// TIA Portal project "Lab1" (V15)

(* hardware
DEVICE "S7-1200 station_1"  S7-1200 Station
   slot 0: "Rack_0"  S7-1200 Rack  Rack  V1.0
   slot 1: "PLC_1"  CPU 1214C AC/DC/Rly  6ES7 214-1BG40-0XB0  V4.2
*)

// ===== PLC "PLC_1"  CPU 1214C AC/DC/Rly =====

VAR_GLOBAL   // PLC tag table "Default tag table"
   "Start_NC" AT %I0.0 : Bool;
   "Manual_NO" AT %I0.2 : Bool;
   "Auto_NO" AT %I0.3 : Bool;
   "Stop_NC" AT %I0.4 : Bool;
   "SigSklop_NC" AT %I0.6 : Bool;
   "Bimetal_NC" AT %I0.7 : Bool;
   "Prekostruj_NO" AT %I1.0 : Bool;
   "Kontaktor_NO" AT %I1.1 : Bool;
   "Zelena" AT %Q0.0 : Bool;
   "Crvena" AT %Q0.1 : Bool;
   "Kontaktor" AT %Q0.2 : Bool;
   "Clock_Byte" AT %MB53 : Byte;
   "Clock_10Hz" AT %M53.0 : Bool;
   "Clock_5Hz" AT %M53.1 : Bool;
   "Clock_2.5Hz" AT %M53.2 : Bool;
   "Clock_2Hz" AT %M53.3 : Bool;
   "Clock_1.25Hz" AT %M53.4 : Bool;
   "Clock_1Hz" AT %M53.5 : Bool;
   "Clock_0.625Hz" AT %M53.6 : Bool;
   "Clock_0.5Hz" AT %M53.7 : Bool;
   "Blink" AT %M3.2 : Bool;
   "Blink_FF" AT %M3.1 : Bool;
   "Blink_Pulse" AT %M3.0 : Bool;
   "Auto_Stanje_FF" AT %M2.0 : Bool;
   "Greska" AT %M0.4 : Bool;
   "Greska_Bimetal" AT %M0.0 : Bool;
   "Greska_Prekostruj" AT %M0.1 : Bool;
   "Greska_Kontaktor" AT %M0.2 : Bool;
   "Greska_Svestop" AT %M0.3 : Bool;
   "Cekamo" AT %M2.2 : Bool;
   "Blink_Cnt_Greska_Pos" AT %M3.3 : Bool;
   "Blink_FF_Greska_Pos" AT %M3.4 : Bool;
   "OFF_NO" AT %M2.1 : Bool;
   "Bimetal_FF" AT %M1.0 : Bool;
   "Prekostruj_FF" AT %M1.1 : Bool;
   "Svestop_FF" AT %M1.3 : Bool;
   "GKontaktor_FF" AT %M1.2 : Bool;
   "Cekamo_Trig_P" AT %M2.3 : Bool;
   "Cekamo_Trig_N" AT %M2.4 : Bool;
   "Ocekivani_Kontaktor" AT %M2.5 : Bool;
END_VAR

// folder: System blocks/Program resources

DATA_BLOCK "Counter_Blink"   // DB1
{ S7_Optimized_Access := 'TRUE' }
AUTHOR : Simatic
FAMILY : IEC
NAME : CNTR
VERSION : 1.0
// stored: InstanceOfName IEC_COUNTER
"IEC_COUNTER"
BEGIN
END_DATA_BLOCK

DATA_BLOCK "Timer_Start"   // DB2
{ S7_Optimized_Access := 'TRUE' }
AUTHOR : Simatic
FAMILY : IEC
NAME : IEC_TMR
VERSION : 1.0
// stored: InstanceOfName IEC_TIMER
"IEC_TIMER"
BEGIN
END_DATA_BLOCK

DATA_BLOCK "Timer_Cekamo"   // DB3
{ S7_Optimized_Access := 'TRUE' }
AUTHOR : Simatic
FAMILY : IEC
NAME : IEC_TMR
VERSION : 1.0
// stored: InstanceOfName IEC_TIMER
"IEC_TIMER"
BEGIN
END_DATA_BLOCK

// folder: (top level)

ORGANIZATION_BLOCK "Main"   // OB1, LAD, ProgramCycle
TITLE = "Main Program Sweep (Cycle)"
{ S7_Optimized_Access := 'TRUE' }
VERSION : 0.1
   VAR_INPUT
      Initial_Call : Bool;   // Initial call of this OB
      Remanence : Bool;   // =True, if remanent data are available
   END_VAR
   VAR_TEMP   // added for the SCL form of the ladder/FBD networks
      _w1 : Bool;
      _w2 : Bool;
      _w3 : Bool;
      _w4 : Bool;
   END_VAR
BEGIN

REGION Network 1: Blink
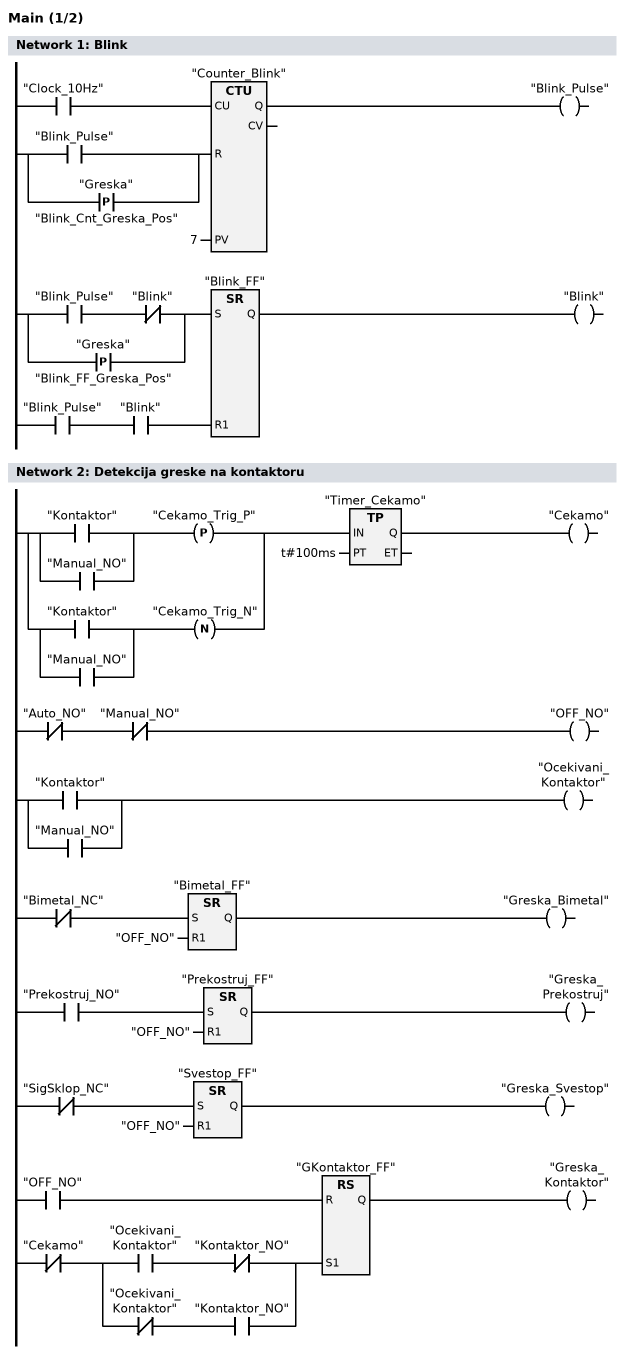
   #_w1 := "Greska" AND NOT "Blink_Cnt_Greska_Pos";   // rising edge of "Greska"
   "Blink_Cnt_Greska_Pos" := "Greska";
   "Counter_Blink".CTU(CU := "Clock_10Hz", R := "Blink_Pulse" OR #_w1, PV := 7);
   "Blink_Pulse" := "Counter_Blink".Q;
   #_w2 := "Greska" AND NOT "Blink_FF_Greska_Pos";   // rising edge of "Greska"
   "Blink_FF_Greska_Pos" := "Greska";
   IF ("Blink_Pulse" AND NOT "Blink") OR #_w2 THEN
       "Blink_FF" := TRUE;   // SR flip-flop
   END_IF;
   IF "Blink_Pulse" AND "Blink" THEN "Blink_FF" := FALSE; END_IF;
   "Blink" := "Blink_FF";
END_REGION

REGION Network 2: Detekcija greske na kontaktoru
   #_w1 := "Kontaktor" OR "Manual_NO";
   #_w2 := #_w1 AND NOT "Cekamo_Trig_P";   // rising edge
   "Cekamo_Trig_P" := #_w1;
   #_w3 := "Kontaktor" OR "Manual_NO";
   #_w4 := NOT #_w3 AND "Cekamo_Trig_N";   // falling edge
   "Cekamo_Trig_N" := #_w3;
   "Timer_Cekamo".TP(IN := #_w2 OR #_w4, PT := t#100ms);
   "Cekamo" := "Timer_Cekamo".Q;
   "OFF_NO" := NOT "Auto_NO" AND NOT "Manual_NO";
   "Ocekivani_Kontaktor" := "Kontaktor" OR "Manual_NO";
   IF NOT "Bimetal_NC" THEN
       "Bimetal_FF" := TRUE;   // SR flip-flop
   END_IF;
   IF "OFF_NO" THEN "Bimetal_FF" := FALSE; END_IF;
   "Greska_Bimetal" := "Bimetal_FF";
   IF "Prekostruj_NO" THEN
       "Prekostruj_FF" := TRUE;   // SR flip-flop
   END_IF;
   IF "OFF_NO" THEN "Prekostruj_FF" := FALSE; END_IF;
   "Greska_Prekostruj" := "Prekostruj_FF";
   IF NOT "SigSklop_NC" THEN
       "Svestop_FF" := TRUE;   // SR flip-flop
   END_IF;
   IF "OFF_NO" THEN "Svestop_FF" := FALSE; END_IF;
   "Greska_Svestop" := "Svestop_FF";
   IF "OFF_NO" THEN
       "GKontaktor_FF" := FALSE;   // RS flip-flop
   END_IF;
   IF NOT "Cekamo" AND (("Ocekivani_Kontaktor" AND NOT "Kontaktor_NO") OR (NOT "Ocekivani_Kontaktor" AND "Kontaktor_NO")) THEN
       "GKontaktor_FF" := TRUE;
   END_IF;
   "Greska_Kontaktor" := "GKontaktor_FF";
END_REGION

REGION Network 3: Formiranje signala greske
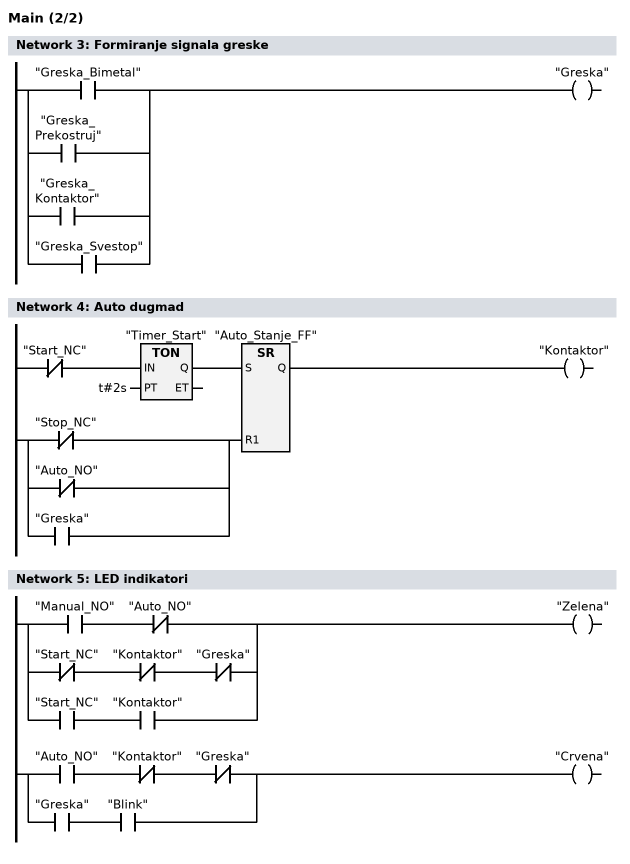
   RUNG wire#powerrail
      Contact( "Greska_Bimetal" )
      wire#w1
      Coil( "Greska" )
   END_RUNG
   RUNG wire#powerrail
      Contact( "Greska_Prekostruj" )
   END_RUNG wire#w1
   RUNG wire#powerrail
      Contact( "Greska_Kontaktor" )
   END_RUNG wire#w1
   RUNG wire#powerrail
      Contact( "Greska_Svestop" )
   END_RUNG wire#w1
   // the same network as SCL:
   "Greska" := "Greska_Bimetal" OR "Greska_Prekostruj" OR "Greska_Kontaktor" OR "Greska_Svestop";
END_REGION

REGION Network 4: Auto dugmad
   "Timer_Start".TON(IN := NOT "Start_NC", PT := t#2s);
   IF "Timer_Start".Q THEN
       "Auto_Stanje_FF" := TRUE;   // SR flip-flop
   END_IF;
   IF NOT "Stop_NC" OR NOT "Auto_NO" OR "Greska" THEN "Auto_Stanje_FF" := FALSE; END_IF;
   "Kontaktor" := "Auto_Stanje_FF";
END_REGION

REGION Network 5: LED indikatori
   RUNG wire#powerrail
      Contact( "Manual_NO" )
      I_Contact( "Auto_NO" )
      wire#w1
      Coil( "Zelena" )
   END_RUNG
   RUNG wire#powerrail
      I_Contact( "Start_NC" )
      I_Contact( "Kontaktor" )
      I_Contact( "Greska" )
   END_RUNG wire#w1
   RUNG wire#powerrail
      Contact( "Start_NC" )
      Contact( "Kontaktor" )
   END_RUNG wire#w1
   RUNG wire#powerrail
      Contact( "Auto_NO" )
      I_Contact( "Kontaktor" )
      I_Contact( "Greska" )
      wire#w2
      Coil( "Crvena" )
   END_RUNG
   RUNG wire#powerrail
      Contact( "Greska" )
      Contact( "Blink" )
   END_RUNG wire#w2
   // the same network as SCL:
   "Zelena" := ("Manual_NO" AND NOT "Auto_NO") OR (NOT "Start_NC" AND NOT "Kontaktor" AND NOT "Greska") OR ("Start_NC" AND "Kontaktor");
   "Crvena" := ("Auto_NO" AND NOT "Kontaktor" AND NOT "Greska") OR ("Greska" AND "Blink");
END_REGION
END_ORGANIZATION_BLOCK